KUKA KRL program: trabalho_concluido.src

&ACCESS RVP3
&REL 2
&PARAM TEMPLATE = C:\KRC\Roboter\Template\vorgabe
&PARAM EDITMASK = *
DEF trabalho_concluido( )
;FOLD ; ;%{PE}%R 4.1.16,%MKUKATPBASIS,%CCOMMENT,%VNORMAL,%P 2:
;ENDFOLD
;FOLD ; Robo 2;%{PE}%R 4.1.16,%MKUKATPBASIS,%CCOMMENT,%VNORMAL,%P 2:Robo 2
;ENDFOLD
;FOLD ; Fim do Processo de Solda;%{PE}%R 4.1.16,%MKUKATPBASIS,%CCOMMENT,%VNORMAL,%P 2:Fim do Processo de Solda
;ENDFOLD
;FOLD ; ;%{PE}%R 4.1.16,%MKUKATPBASIS,%CCOMMENT,%VNORMAL,%P 2:
;ENDFOLD
;FOLD PULSE 3333 'R2_Trabalho Concluido' State=TRUE CONT Time=3 sec;%{PE}%R 8.2.20,%MKUKATPBASIS,%COUT,%VPULSE,%P 2:3333, 3:R2_Trabalho Concluido, 5:TRUE, 6:CONTINUE, 8:3
CONTINUE
PULSE($OUT[3333], TRUE,3)
;ENDFOLD

END
